// TIA Portal V15.1 export
// export: Created 2020-06-12T07:35:48.1005859Z, ExportSetting None, DisplayName Totally Integrated Automation Portal, DisplayVersion V15.1, DisplayName TIA Portal Openness, DisplayVersion V15.1, DisplayName STEP 7 Professional, DisplayVersion V15.1, DisplayName STEP 7 Safety, DisplayVersion V15.1, DisplayName WinCC Advanced, DisplayVersion V15.1
FUNCTION "PWR_pfc" : Void   // FC114, FBD
TITLE = Power factor correction
{ S7_Optimized_Access := 'TRUE' }
// stored: SetENOAutomatically False
   VAR_TEMP
      _csf : Bool;   // Common system fault
      _on : Bool;
      _auto_on1 : Bool;
      _auto_on2 : Bool;
      _auto_on3 : Bool;
      _auto_on4 : Bool;
      _auto_on5 : Bool;
      _auto_on6 : Bool;
      _auto_off1 : Bool;
      _auto_off2 : Bool;
      _auto_off3 : Bool;
      _auto_off4 : Bool;
      _auto_off5 : Bool;
      _auto_off6 : Bool;
      _lock_time : Time;   // Capacitor discharging time
      _num_set : Int;
      _num_act : Int;
      tAppPower : Real;
      tActPower : Real;
      tActVoltage : Real;
      tActCurrent : Real;
      tIson1 : Bool;
      tIson2 : Bool;
      tIson3 : Bool;
      tIson4 : Bool;
      tIson5 : Bool;
      tIson6 : Bool;
      tIson7 : Bool;
      tIson8 : Bool;
      _filt_time : Time;
      tAutoEn : Bool;
      tVolatgePrim : Real;
      tCosPhi : Real;
      tSPowerPrim : Real;
      tQPowerPrim : Real;
      tReqPfcOn : Bool;
      tReqPfcOff : Bool;
      tReqPfcMan : Bool;
      tReqPfcAuto : Bool;
   END_VAR
BEGIN

REGION Network 1: Common System Fault
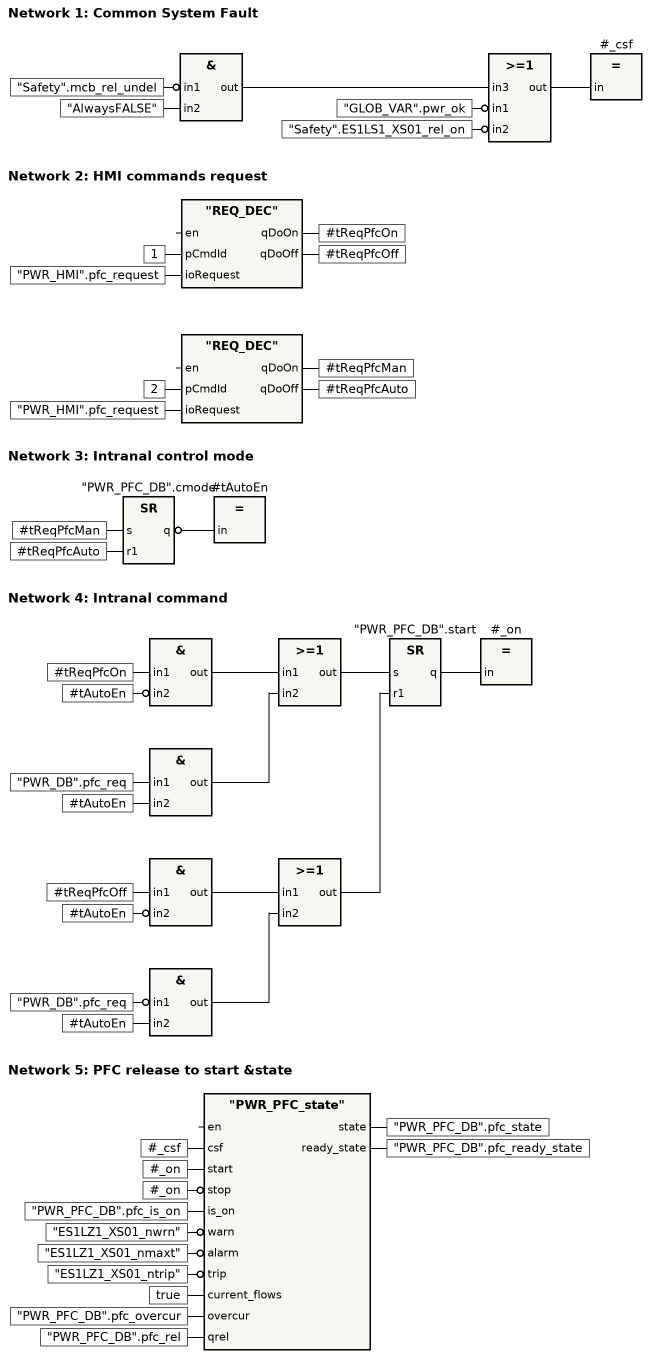
   #_csf := (NOT "Safety".mcb_rel_undel AND "AlwaysFALSE") OR NOT "GLOB_VAR".pwr_ok OR NOT "Safety".ES1LS1_XS01_rel_on;
END_REGION

REGION Network 2: HMI commands request
   "REQ_DEC"(pCmdId := 1, ioRequest := "PWR_HMI".pfc_request, qDoOn => #tReqPfcOn, qDoOff => #tReqPfcOff);
   "REQ_DEC"(pCmdId := 2, ioRequest := "PWR_HMI".pfc_request, qDoOn => #tReqPfcMan, qDoOff => #tReqPfcAuto);
END_REGION

REGION Network 3: Intranal control mode
   IF #tReqPfcMan THEN
       "PWR_PFC_DB".cmode := TRUE;   // SR flip-flop
   END_IF;
   IF #tReqPfcAuto THEN "PWR_PFC_DB".cmode := FALSE; END_IF;
   #tAutoEn := NOT "PWR_PFC_DB".cmode;
END_REGION

REGION Network 4: Intranal command
   IF (#tReqPfcOn AND NOT #tAutoEn) OR ("PWR_DB".pfc_req AND #tAutoEn) THEN
       "PWR_PFC_DB".start := TRUE;   // SR flip-flop
   END_IF;
   IF (#tReqPfcOff AND NOT #tAutoEn) OR (NOT "PWR_DB".pfc_req AND #tAutoEn) THEN
       "PWR_PFC_DB".start := FALSE;
   END_IF;
   #_on := "PWR_PFC_DB".start;
END_REGION

REGION Network 5: PFC release to start &state
   // REMOVED "PWR_DB".current_flow
   "PWR_PFC_state"(csf := #_csf,
                   start := #_on,
                   stop := NOT #_on,
                   is_on := "PWR_PFC_DB".pfc_is_on,
                   warn := NOT "ES1LZ1_XS01_nwrn",
                   alarm := NOT "ES1LZ1_XS01_nmaxt",
                   trip := NOT "ES1LZ1_XS01_ntrip",
                   current_flows := true,
                   overcur := "PWR_PFC_DB".pfc_overcur,
                   qrel := "PWR_PFC_DB".pfc_rel,
                   state => "PWR_PFC_DB".pfc_state,
                   ready_state => "PWR_PFC_DB".pfc_ready_state);
END_REGION

REGION Network 6: HMI status
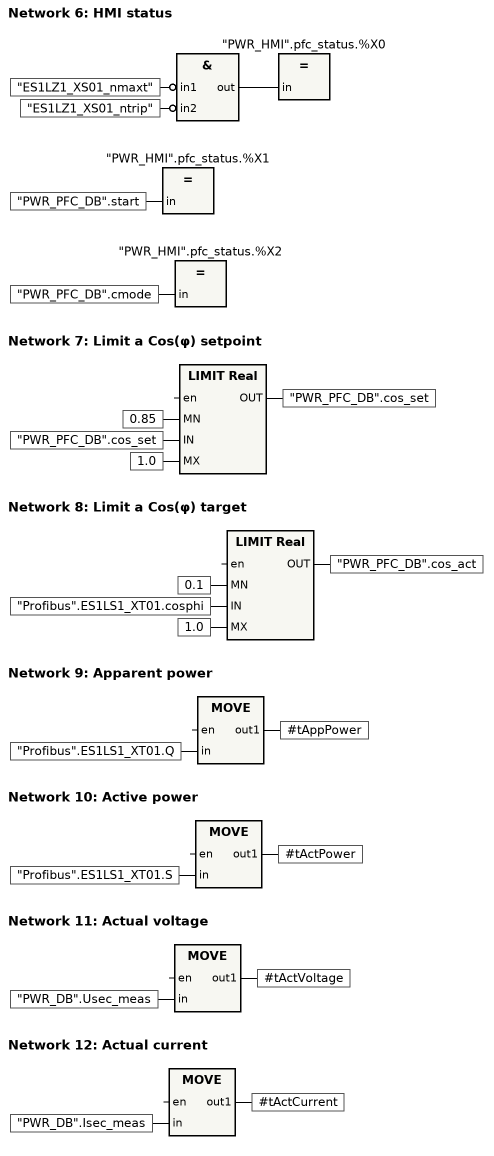
   "PWR_HMI".pfc_status.%X0 := NOT "ES1LZ1_XS01_nmaxt" AND NOT "ES1LZ1_XS01_ntrip";
   "PWR_HMI".pfc_status.%X1 := "PWR_PFC_DB".start;
   "PWR_HMI".pfc_status.%X2 := "PWR_PFC_DB".cmode;
END_REGION

REGION Network 7: Limit a Cos(φ) setpoint
   "PWR_PFC_DB".cos_set := LIMIT(MN := 0.85, IN := "PWR_PFC_DB".cos_set, MX := 1.0);
END_REGION

REGION Network 8: Limit a Cos(φ) target
   "PWR_PFC_DB".cos_act := LIMIT(MN := 0.1, IN := "Profibus".ES1LS1_XT01.cosphi, MX := 1.0);
END_REGION

REGION Network 9: Apparent power
   #tAppPower := "Profibus".ES1LS1_XT01.Q;
END_REGION

REGION Network 10: Active power
   #tActPower := "Profibus".ES1LS1_XT01.S;
END_REGION

REGION Network 11: Actual voltage
   #tActVoltage := "PWR_DB".Usec_meas;
END_REGION

REGION Network 12: Actual current
   #tActCurrent := "PWR_DB".Isec_meas;
END_REGION

REGION Network 13: Filter: Cos(Phi)
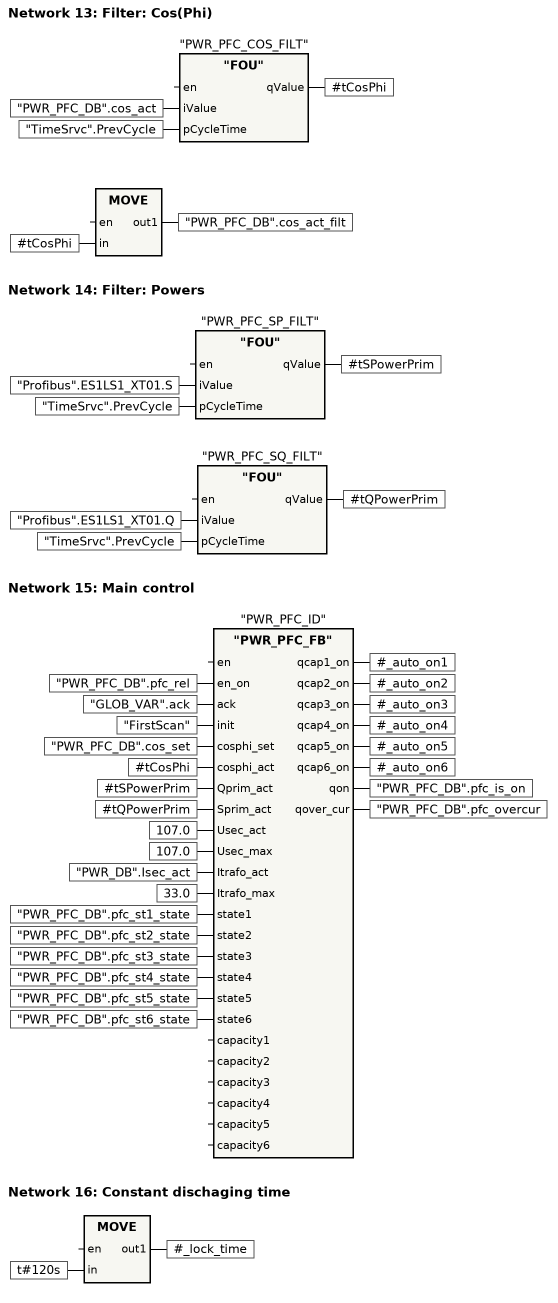
   "PWR_PFC_COS_FILT"(iValue := "PWR_PFC_DB".cos_act, pCycleTime := "TimeSrvc".PrevCycle, qValue => #tCosPhi);   // "FOU"
   "PWR_PFC_DB".cos_act_filt := #tCosPhi;
END_REGION

REGION Network 14: Filter: Powers
   "PWR_PFC_SP_FILT"(iValue := "Profibus".ES1LS1_XT01.S,   // "FOU"
                     pCycleTime := "TimeSrvc".PrevCycle,
                     qValue => #tSPowerPrim);
   "PWR_PFC_SQ_FILT"(iValue := "Profibus".ES1LS1_XT01.Q,   // "FOU"
                     pCycleTime := "TimeSrvc".PrevCycle,
                     qValue => #tQPowerPrim);
END_REGION

REGION Network 15: Main control
   // DEBUG: #tQPowerPrim <-> #tSPowerPrim
   "PWR_PFC_ID"(en_on := "PWR_PFC_DB".pfc_rel,   // "PWR_PFC_FB"
                ack := "GLOB_VAR".ack,
                init := "FirstScan",
                cosphi_set := "PWR_PFC_DB".cos_set,
                cosphi_act := #tCosPhi,
                Qprim_act := #tSPowerPrim,
                Sprim_act := #tQPowerPrim,
                Usec_act := 107.0,
                Usec_max := 107.0,
                Itrafo_act := "PWR_DB".Isec_act,
                Itrafo_max := 33.0,
                state1 := "PWR_PFC_DB".pfc_st1_state,
                state2 := "PWR_PFC_DB".pfc_st2_state,
                state3 := "PWR_PFC_DB".pfc_st3_state,
                state4 := "PWR_PFC_DB".pfc_st4_state,
                state5 := "PWR_PFC_DB".pfc_st5_state,
                state6 := "PWR_PFC_DB".pfc_st6_state,
                qcap1_on => #_auto_on1,
                qcap2_on => #_auto_on2,
                qcap3_on => #_auto_on3,
                qcap4_on => #_auto_on4,
                qcap5_on => #_auto_on5,
                qcap6_on => #_auto_on6,
                qon => "PWR_PFC_DB".pfc_is_on,
                qover_cur => "PWR_PFC_DB".pfc_overcur);
END_REGION

REGION Network 16: Constant dischaging time
   #_lock_time := t#120s;
END_REGION

REGION Network 17: feddback filter time
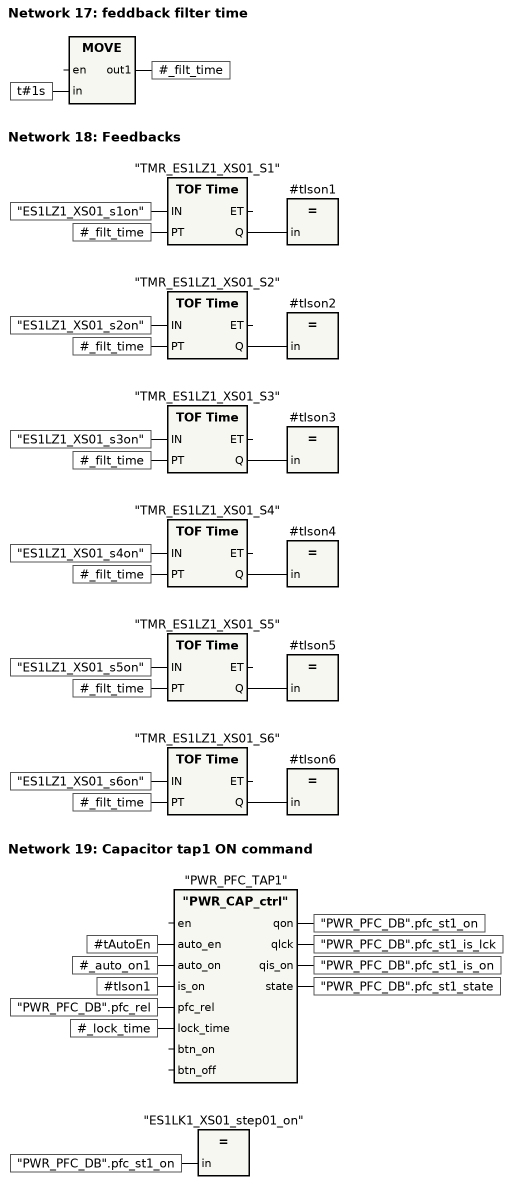
   #_filt_time := t#1s;
END_REGION

REGION Network 18: Feedbacks
   "TMR_ES1LZ1_XS01_S1".TOF(IN := "ES1LZ1_XS01_s1on", PT := #_filt_time);
   #tIson1 := "TMR_ES1LZ1_XS01_S1".Q;
   "TMR_ES1LZ1_XS01_S2".TOF(IN := "ES1LZ1_XS01_s2on", PT := #_filt_time);
   #tIson2 := "TMR_ES1LZ1_XS01_S2".Q;
   "TMR_ES1LZ1_XS01_S3".TOF(IN := "ES1LZ1_XS01_s3on", PT := #_filt_time);
   #tIson3 := "TMR_ES1LZ1_XS01_S3".Q;
   "TMR_ES1LZ1_XS01_S4".TOF(IN := "ES1LZ1_XS01_s4on", PT := #_filt_time);
   #tIson4 := "TMR_ES1LZ1_XS01_S4".Q;
   "TMR_ES1LZ1_XS01_S5".TOF(IN := "ES1LZ1_XS01_s5on", PT := #_filt_time);
   #tIson5 := "TMR_ES1LZ1_XS01_S5".Q;
   "TMR_ES1LZ1_XS01_S6".TOF(IN := "ES1LZ1_XS01_s6on", PT := #_filt_time);
   #tIson6 := "TMR_ES1LZ1_XS01_S6".Q;
END_REGION

REGION Network 19: Capacitor tap1 ON command
   "PWR_PFC_TAP1"(auto_en := #tAutoEn,   // "PWR_CAP_ctrl"
                  auto_on := #_auto_on1,
                  is_on := #tIson1,
                  pfc_rel := "PWR_PFC_DB".pfc_rel,
                  lock_time := #_lock_time,
                  qon => "PWR_PFC_DB".pfc_st1_on,
                  qlck => "PWR_PFC_DB".pfc_st1_is_lck,
                  qis_on => "PWR_PFC_DB".pfc_st1_is_on,
                  state => "PWR_PFC_DB".pfc_st1_state);
   "ES1LK1_XS01_step01_on" := "PWR_PFC_DB".pfc_st1_on;
END_REGION

REGION Network 20: Capacitor tap2 ON command
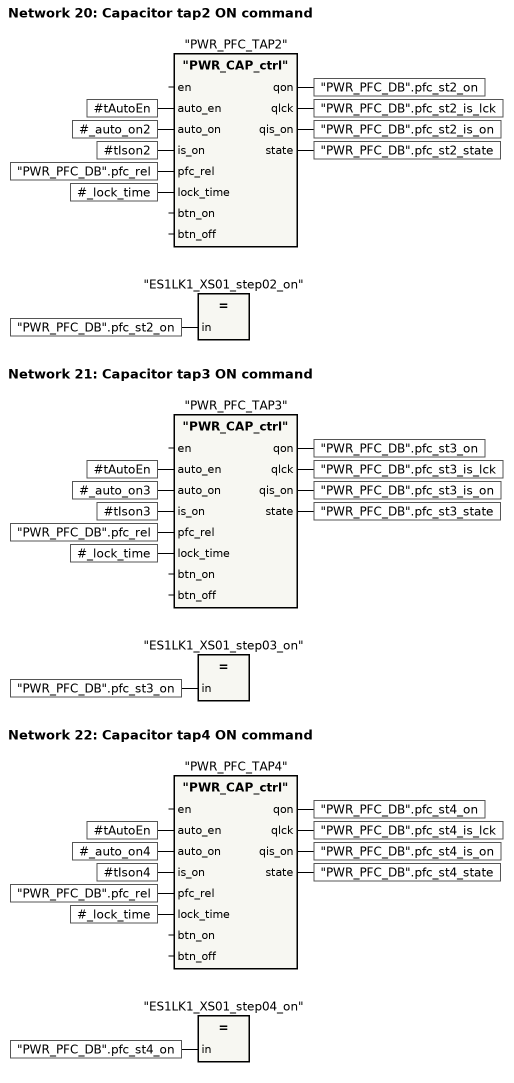
   "PWR_PFC_TAP2"(auto_en := #tAutoEn,   // "PWR_CAP_ctrl"
                  auto_on := #_auto_on2,
                  is_on := #tIson2,
                  pfc_rel := "PWR_PFC_DB".pfc_rel,
                  lock_time := #_lock_time,
                  qon => "PWR_PFC_DB".pfc_st2_on,
                  qlck => "PWR_PFC_DB".pfc_st2_is_lck,
                  qis_on => "PWR_PFC_DB".pfc_st2_is_on,
                  state => "PWR_PFC_DB".pfc_st2_state);
   "ES1LK1_XS01_step02_on" := "PWR_PFC_DB".pfc_st2_on;
END_REGION

REGION Network 21: Capacitor tap3 ON command
   "PWR_PFC_TAP3"(auto_en := #tAutoEn,   // "PWR_CAP_ctrl"
                  auto_on := #_auto_on3,
                  is_on := #tIson3,
                  pfc_rel := "PWR_PFC_DB".pfc_rel,
                  lock_time := #_lock_time,
                  qon => "PWR_PFC_DB".pfc_st3_on,
                  qlck => "PWR_PFC_DB".pfc_st3_is_lck,
                  qis_on => "PWR_PFC_DB".pfc_st3_is_on,
                  state => "PWR_PFC_DB".pfc_st3_state);
   "ES1LK1_XS01_step03_on" := "PWR_PFC_DB".pfc_st3_on;
END_REGION

REGION Network 22: Capacitor tap4 ON command
   "PWR_PFC_TAP4"(auto_en := #tAutoEn,   // "PWR_CAP_ctrl"
                  auto_on := #_auto_on4,
                  is_on := #tIson4,
                  pfc_rel := "PWR_PFC_DB".pfc_rel,
                  lock_time := #_lock_time,
                  qon => "PWR_PFC_DB".pfc_st4_on,
                  qlck => "PWR_PFC_DB".pfc_st4_is_lck,
                  qis_on => "PWR_PFC_DB".pfc_st4_is_on,
                  state => "PWR_PFC_DB".pfc_st4_state);
   "ES1LK1_XS01_step04_on" := "PWR_PFC_DB".pfc_st4_on;
END_REGION

REGION Network 23: Capacitor tap5 ON command
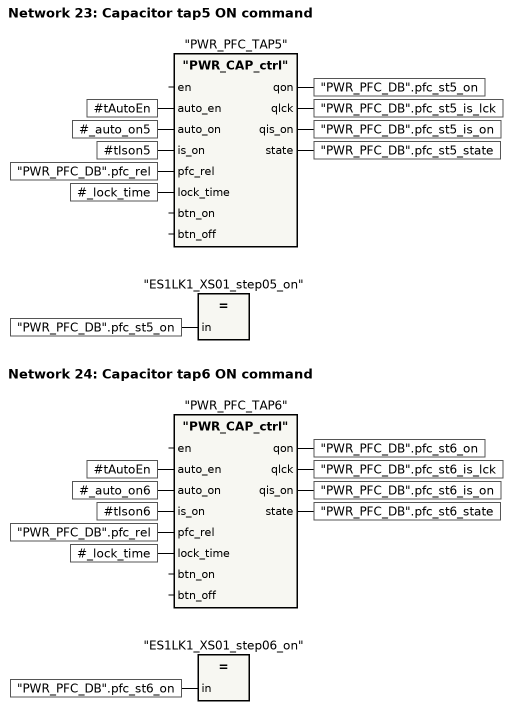
   "PWR_PFC_TAP5"(auto_en := #tAutoEn,   // "PWR_CAP_ctrl"
                  auto_on := #_auto_on5,
                  is_on := #tIson5,
                  pfc_rel := "PWR_PFC_DB".pfc_rel,
                  lock_time := #_lock_time,
                  qon => "PWR_PFC_DB".pfc_st5_on,
                  qlck => "PWR_PFC_DB".pfc_st5_is_lck,
                  qis_on => "PWR_PFC_DB".pfc_st5_is_on,
                  state => "PWR_PFC_DB".pfc_st5_state);
   "ES1LK1_XS01_step05_on" := "PWR_PFC_DB".pfc_st5_on;
END_REGION

REGION Network 24: Capacitor tap6 ON command
   "PWR_PFC_TAP6"(auto_en := #tAutoEn,   // "PWR_CAP_ctrl"
                  auto_on := #_auto_on6,
                  is_on := #tIson6,
                  pfc_rel := "PWR_PFC_DB".pfc_rel,
                  lock_time := #_lock_time,
                  qon => "PWR_PFC_DB".pfc_st6_on,
                  qlck => "PWR_PFC_DB".pfc_st6_is_lck,
                  qis_on => "PWR_PFC_DB".pfc_st6_is_on,
                  state => "PWR_PFC_DB".pfc_st6_state);
   "ES1LK1_XS01_step06_on" := "PWR_PFC_DB".pfc_st6_on;
END_REGION

REGION Network 25: Number of Capacitor switched ON
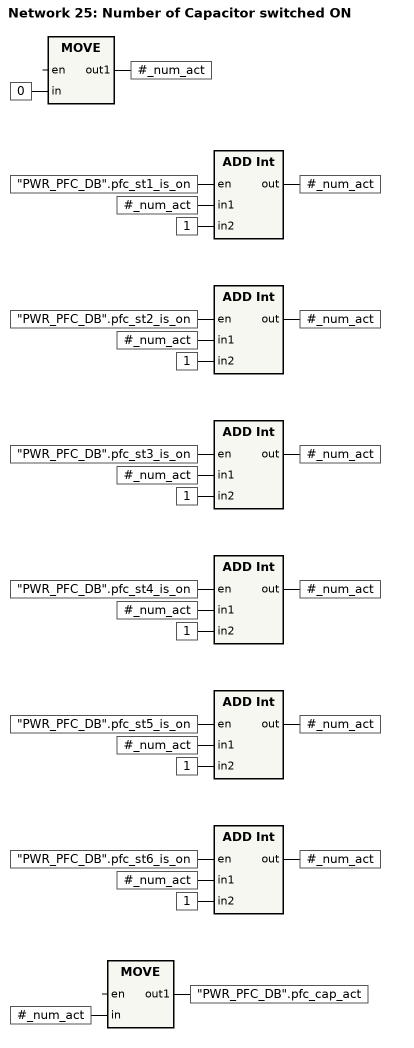
   #_num_act := 0;
   IF "PWR_PFC_DB".pfc_st1_is_on THEN #_num_act := #_num_act + 1; END_IF;
   IF "PWR_PFC_DB".pfc_st2_is_on THEN #_num_act := #_num_act + 1; END_IF;
   IF "PWR_PFC_DB".pfc_st3_is_on THEN #_num_act := #_num_act + 1; END_IF;
   IF "PWR_PFC_DB".pfc_st4_is_on THEN #_num_act := #_num_act + 1; END_IF;
   IF "PWR_PFC_DB".pfc_st5_is_on THEN #_num_act := #_num_act + 1; END_IF;
   IF "PWR_PFC_DB".pfc_st6_is_on THEN #_num_act := #_num_act + 1; END_IF;
   "PWR_PFC_DB".pfc_cap_act := #_num_act;
END_REGION

REGION Network 26: Number of Capacitor set ON
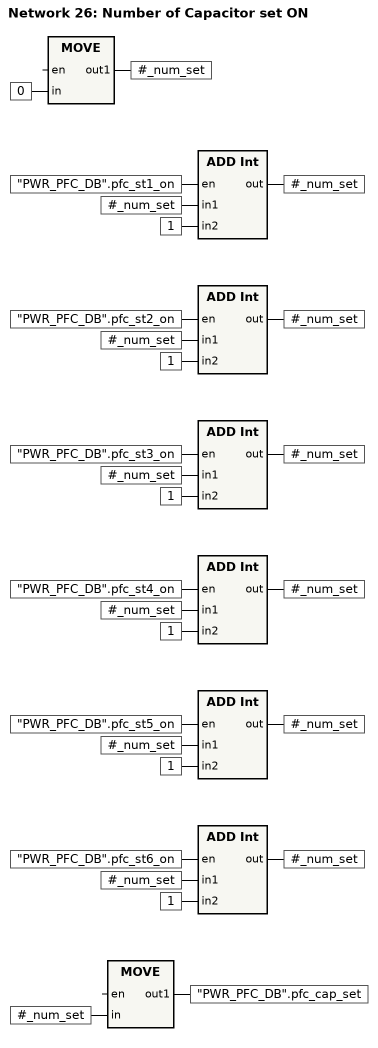
   #_num_set := 0;
   IF "PWR_PFC_DB".pfc_st1_on THEN #_num_set := #_num_set + 1; END_IF;
   IF "PWR_PFC_DB".pfc_st2_on THEN #_num_set := #_num_set + 1; END_IF;
   IF "PWR_PFC_DB".pfc_st3_on THEN #_num_set := #_num_set + 1; END_IF;
   IF "PWR_PFC_DB".pfc_st4_on THEN #_num_set := #_num_set + 1; END_IF;
   IF "PWR_PFC_DB".pfc_st5_on THEN #_num_set := #_num_set + 1; END_IF;
   IF "PWR_PFC_DB".pfc_st6_on THEN #_num_set := #_num_set + 1; END_IF;
   "PWR_PFC_DB".pfc_cap_set := #_num_set;
END_REGION
END_FUNCTION
